// TIA Portal V18 export
DATA_BLOCK "Calculations_DB"   // DB10
// stored: AutoNumber false, InstanceOfName Calculations, InstanceOfType FB
"Calculations"
   // VAR
   //    M1_LPF { S7_SetPoint := 'True'} : "LowPassFilter";
   //    M2_LPF { S7_SetPoint := 'True'} : "LowPassFilter";
   //    TDPressFwd_LPF { S7_SetPoint := 'True'} : "LowPassFilter";
   //    TDPressRev_LPF { S7_SetPoint := 'True'} : "LowPassFilter";
   //    ClosedLoopTemp_LPF { S7_SetPoint := 'True'} : "LowPassFilter";
   //    ChargeFlow_LPF { S7_SetPoint := 'True'} : "LowPassFilter";
   //    HotOilFlow_LPF { S7_SetPoint := 'True'} : "LowPassFilter";
   //    AuxFlow_LPF { S7_SetPoint := 'True'} : "LowPassFilter";
   //    ChargePress1_LPF { S7_SetPoint := 'True'} : "LowPassFilter";
   //    ChargePress2_LPF { S7_SetPoint := 'True'} : "LowPassFilter";
   //    DrillTorqPotLPF { S7_SetPoint := 'True'} : "LowPassFilter";
   //    MUTorqPotLPF { S7_SetPoint := 'True'} : "LowPassFilter";
   //    DrillThrottlePotLPF { S7_SetPoint := 'True'} : "LowPassFilter";
   //    ActTorq_LPF { S7_SetPoint := 'True'} : "LowPassFilter";
   //    DrillRecPTO_TP { S7_SetPoint := 'True'} : TP_TIME;
   //    DrillRecMax { S7_SetPoint := 'True'} : Bool;
   // END_VAR
BEGIN
END_DATA_BLOCK
